(* CoDeSys 2.3 export: ST_POWERPACK_CFG.EXP *)

(* Data type *)
TYPE ST_POWERPACK_CFG :
STRUCT
	Hyst_HP : REAL;
	Hyst_LP : REAL;
	Hyst_TM : REAL;	(*Seconds*)

	Thr_HP : REAL;
	Thr_LP : REAL;

	Cycle : REAL;	(*Second*)
END_STRUCT
END_TYPE
